{attribute 'GeneratedUsingTerminal: EK1122-0000-0018'}
{attribute addProperty BoxType "EK1122-0000-0018"}
{attribute addProperty Id "Beckhoff_ER8xxxsub_EK1100EK1100_1FC0878B2A_0001_ER8309_1022_0018ER8309_0B5CA5B162"}
{attribute addProperty CRC "864426720"}
{attribute addProperty Size "64"}
TYPE Beckhoff_ER8xxxEK1122_33861AE0 EXTENDS EK1122_1FC0878B :
STRUCT
	{attribute addProperty Name "Beckhoff_ER8xxxsub_EK1100"}
	{attribute addProperty PreviousPort "Beckhoff ER8xxxEK1122 : D"}
	Beckhoff_ER8xxxsub_EK1100 : EK1100_1FC0878B;
	{attribute addProperty Name "A_0001_ER8309_1022_0018"}
	{attribute addProperty PreviousPort "Beckhoff ER8xxxsub EK1100 : C"}
	A_0001_ER8309_1022_0018 : ER8309_0B5CA5B1;
END_STRUCT
END_TYPE

(* stored: Version 1.2.0.0, ProductVersion 3.1.4024.9
   DUT Beckhoff_ER8xxxEK1122_33861AE0: Id {f567700b-b683-46b7-b56d-710e9393e078} *)
